PROGRAM BasketMemoryCtrl
VAR

	NIL: BOOL;

END_VAR

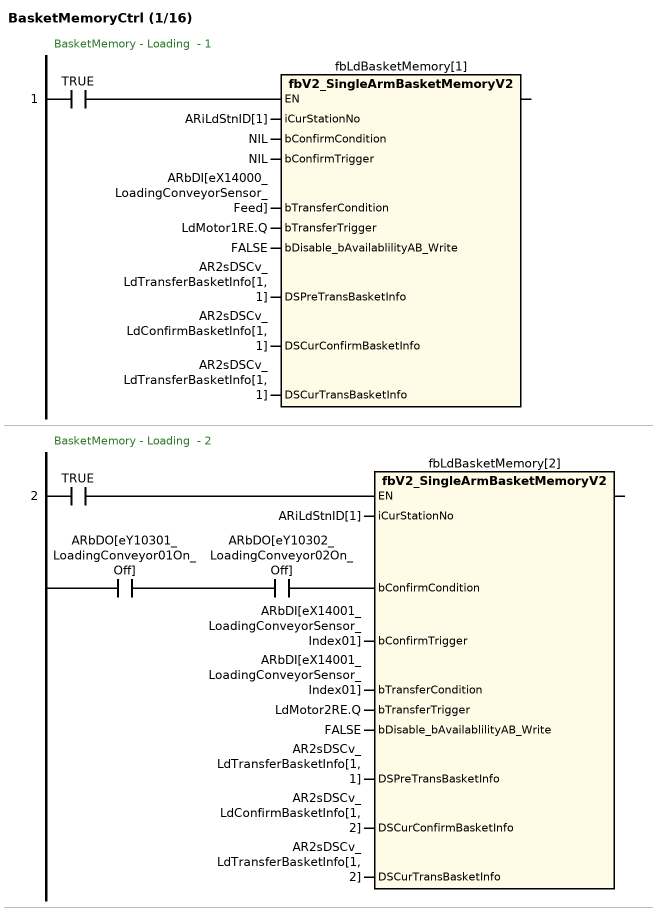
// NETWORK 1
// BasketMemory - Loading  - 1
fbLdBasketMemory[1](
    iCurStationNo := ARiLdStnID[1],
    bConfirmCondition := NIL,
    bConfirmTrigger := NIL,
    bTransferCondition := ARbDI[eX14000_LoadingConveyorSensor_Feed],
    bTransferTrigger := LdMotor1RE.Q,
    bDisable_bAvailablilityAB_Write := FALSE,
    DSPreTransBasketInfo := AR2sDSCv_LdTransferBasketInfo[1,1],
    DSCurConfirmBasketInfo := AR2sDSCv_LdConfirmBasketInfo[1,1],
    DSCurTransBasketInfo := AR2sDSCv_LdTransferBasketInfo[1,1]); // fbV2_SingleArmBasketMemoryV2

// NETWORK 2
// BasketMemory - Loading  - 2
fbLdBasketMemory[2](
    iCurStationNo := ARiLdStnID[1],
    bConfirmCondition := ARbDO[eY10301_LoadingConveyor01On_Off] AND ARbDO[eY10302_LoadingConveyor02On_Off],
    bConfirmTrigger := ARbDI[eX14001_LoadingConveyorSensor_Index01],
    bTransferCondition := ARbDI[eX14001_LoadingConveyorSensor_Index01],
    bTransferTrigger := LdMotor2RE.Q,
    bDisable_bAvailablilityAB_Write := FALSE,
    DSPreTransBasketInfo := AR2sDSCv_LdTransferBasketInfo[1,1],
    DSCurConfirmBasketInfo := AR2sDSCv_LdConfirmBasketInfo[1,2],
    DSCurTransBasketInfo := AR2sDSCv_LdTransferBasketInfo[1,2]); // fbV2_SingleArmBasketMemoryV2

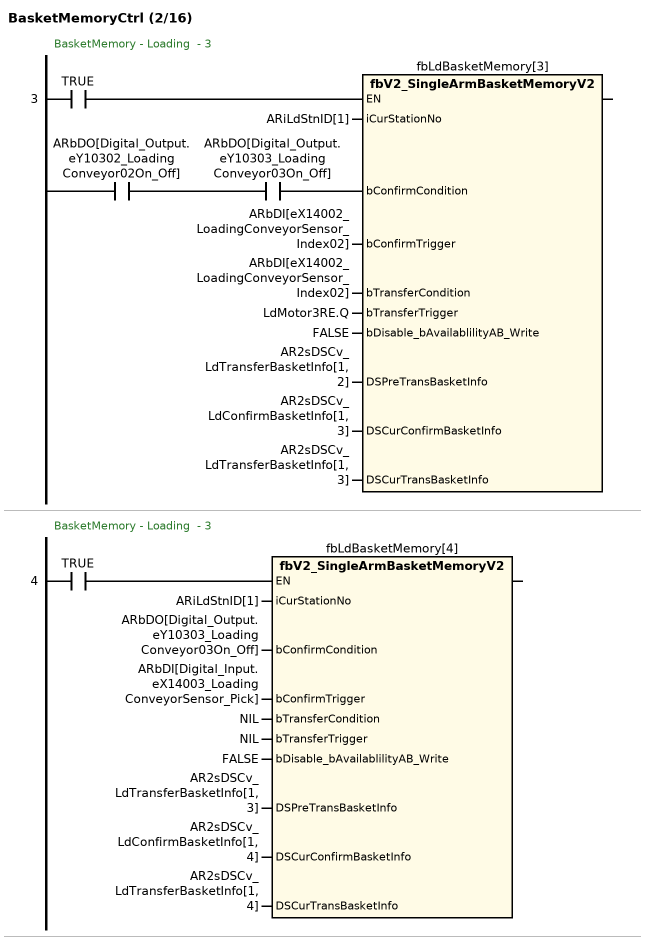
// NETWORK 3
// BasketMemory - Loading  - 3
fbLdBasketMemory[3](
    iCurStationNo := ARiLdStnID[1],
    bConfirmCondition := ARbDO[Digital_Output.eY10302_LoadingConveyor02On_Off] AND ARbDO[Digital_Output.eY10303_LoadingConveyor03On_Off],
    bConfirmTrigger := ARbDI[eX14002_LoadingConveyorSensor_Index02],
    bTransferCondition := ARbDI[eX14002_LoadingConveyorSensor_Index02],
    bTransferTrigger := LdMotor3RE.Q,
    bDisable_bAvailablilityAB_Write := FALSE,
    DSPreTransBasketInfo := AR2sDSCv_LdTransferBasketInfo[1,2],
    DSCurConfirmBasketInfo := AR2sDSCv_LdConfirmBasketInfo[1,3],
    DSCurTransBasketInfo := AR2sDSCv_LdTransferBasketInfo[1,3]); // fbV2_SingleArmBasketMemoryV2

// NETWORK 4
// BasketMemory - Loading  - 3
fbLdBasketMemory[4](
    iCurStationNo := ARiLdStnID[1],
    bConfirmCondition := ARbDO[Digital_Output.eY10303_LoadingConveyor03On_Off],
    bConfirmTrigger := ARbDI[Digital_Input.eX14003_LoadingConveyorSensor_Pick],
    bTransferCondition := NIL,
    bTransferTrigger := NIL,
    bDisable_bAvailablilityAB_Write := FALSE,
    DSPreTransBasketInfo := AR2sDSCv_LdTransferBasketInfo[1,3],
    DSCurConfirmBasketInfo := AR2sDSCv_LdConfirmBasketInfo[1,4],
    DSCurTransBasketInfo := AR2sDSCv_LdTransferBasketInfo[1,4]); // fbV2_SingleArmBasketMemoryV2

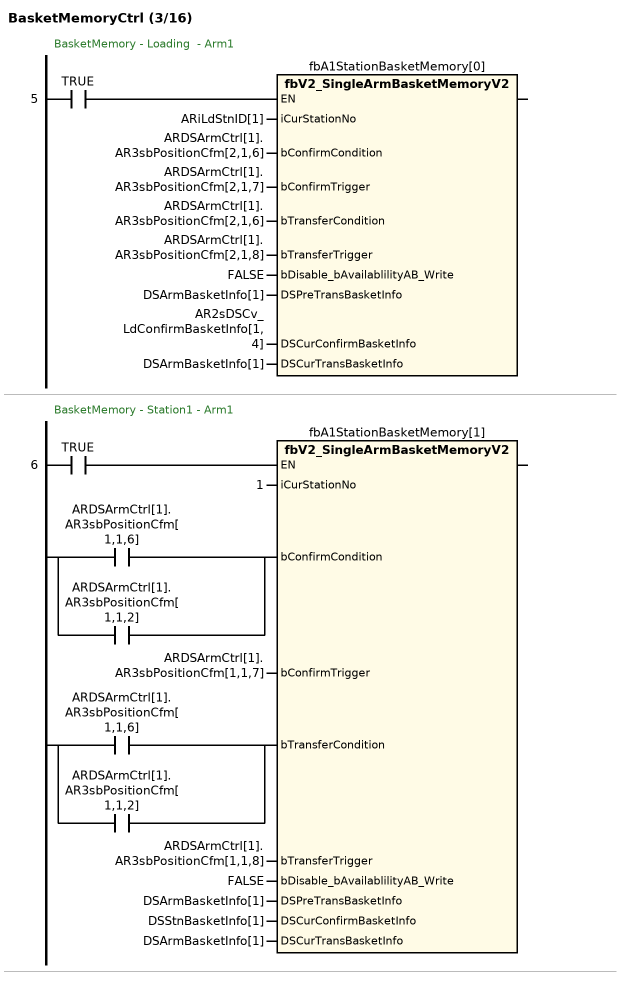
// NETWORK 5
// BasketMemory - Loading  - Arm1
fbA1StationBasketMemory[0](
    iCurStationNo := ARiLdStnID[1],
    bConfirmCondition := ARDSArmCtrl[1].AR3sbPositionCfm[2,1,6],
    bConfirmTrigger := ARDSArmCtrl[1].AR3sbPositionCfm[2,1,7],
    bTransferCondition := ARDSArmCtrl[1].AR3sbPositionCfm[2,1,6],
    bTransferTrigger := ARDSArmCtrl[1].AR3sbPositionCfm[2,1,8],
    bDisable_bAvailablilityAB_Write := FALSE,
    DSPreTransBasketInfo := DSArmBasketInfo[1],
    DSCurConfirmBasketInfo := AR2sDSCv_LdConfirmBasketInfo[1,4],
    DSCurTransBasketInfo := DSArmBasketInfo[1]); // fbV2_SingleArmBasketMemoryV2

// NETWORK 6
// BasketMemory - Station1 - Arm1
fbA1StationBasketMemory[1](
    iCurStationNo := 1,
    bConfirmCondition := ARDSArmCtrl[1].AR3sbPositionCfm[1,1,6] OR ARDSArmCtrl[1].AR3sbPositionCfm[1,1,2],
    bConfirmTrigger := ARDSArmCtrl[1].AR3sbPositionCfm[1,1,7],
    bTransferCondition := ARDSArmCtrl[1].AR3sbPositionCfm[1,1,6] OR ARDSArmCtrl[1].AR3sbPositionCfm[1,1,2],
    bTransferTrigger := ARDSArmCtrl[1].AR3sbPositionCfm[1,1,8],
    bDisable_bAvailablilityAB_Write := FALSE,
    DSPreTransBasketInfo := DSArmBasketInfo[1],
    DSCurConfirmBasketInfo := DSStnBasketInfo[1],
    DSCurTransBasketInfo := DSArmBasketInfo[1]); // fbV2_SingleArmBasketMemoryV2

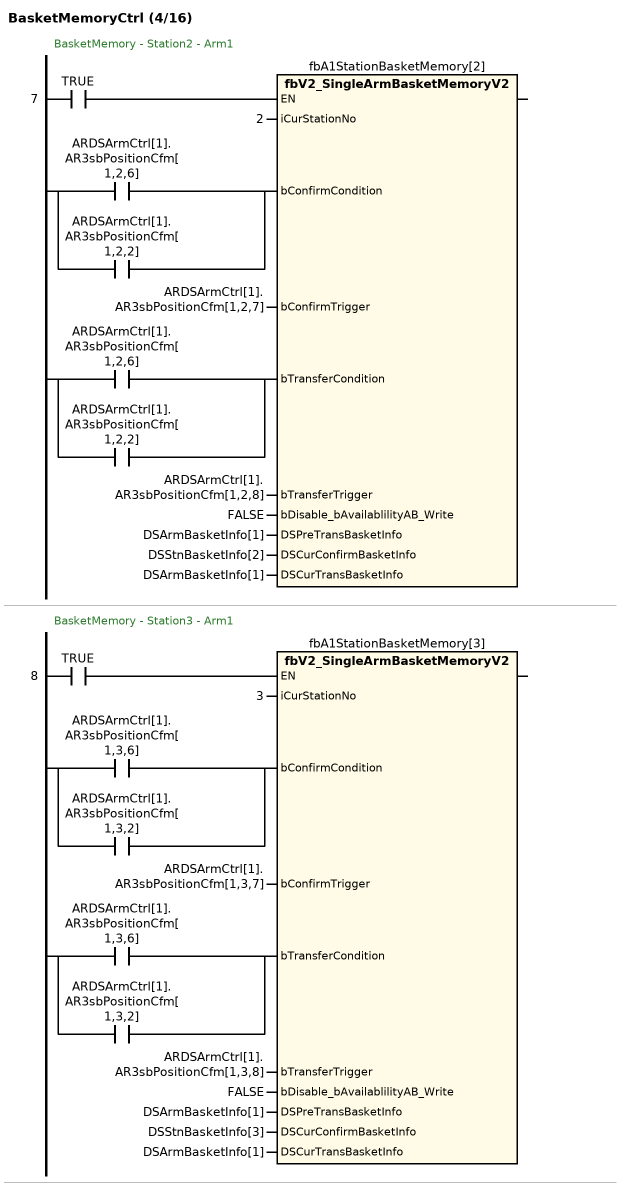
// NETWORK 7
// BasketMemory - Station2 - Arm1
fbA1StationBasketMemory[2](
    iCurStationNo := 2,
    bConfirmCondition := ARDSArmCtrl[1].AR3sbPositionCfm[1,2,6] OR ARDSArmCtrl[1].AR3sbPositionCfm[1,2,2],
    bConfirmTrigger := ARDSArmCtrl[1].AR3sbPositionCfm[1,2,7],
    bTransferCondition := ARDSArmCtrl[1].AR3sbPositionCfm[1,2,6] OR ARDSArmCtrl[1].AR3sbPositionCfm[1,2,2],
    bTransferTrigger := ARDSArmCtrl[1].AR3sbPositionCfm[1,2,8],
    bDisable_bAvailablilityAB_Write := FALSE,
    DSPreTransBasketInfo := DSArmBasketInfo[1],
    DSCurConfirmBasketInfo := DSStnBasketInfo[2],
    DSCurTransBasketInfo := DSArmBasketInfo[1]); // fbV2_SingleArmBasketMemoryV2

// NETWORK 8
// BasketMemory - Station3 - Arm1
fbA1StationBasketMemory[3](
    iCurStationNo := 3,
    bConfirmCondition := ARDSArmCtrl[1].AR3sbPositionCfm[1,3,6] OR ARDSArmCtrl[1].AR3sbPositionCfm[1,3,2],
    bConfirmTrigger := ARDSArmCtrl[1].AR3sbPositionCfm[1,3,7],
    bTransferCondition := ARDSArmCtrl[1].AR3sbPositionCfm[1,3,6] OR ARDSArmCtrl[1].AR3sbPositionCfm[1,3,2],
    bTransferTrigger := ARDSArmCtrl[1].AR3sbPositionCfm[1,3,8],
    bDisable_bAvailablilityAB_Write := FALSE,
    DSPreTransBasketInfo := DSArmBasketInfo[1],
    DSCurConfirmBasketInfo := DSStnBasketInfo[3],
    DSCurTransBasketInfo := DSArmBasketInfo[1]); // fbV2_SingleArmBasketMemoryV2

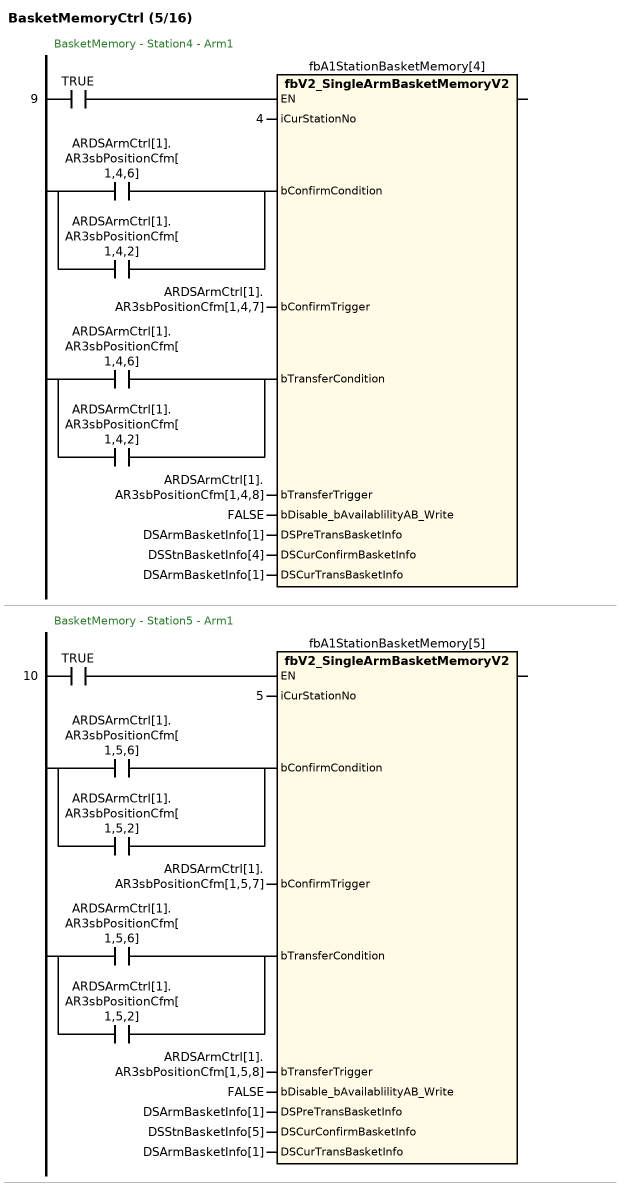
// NETWORK 9
// BasketMemory - Station4 - Arm1
fbA1StationBasketMemory[4](
    iCurStationNo := 4,
    bConfirmCondition := ARDSArmCtrl[1].AR3sbPositionCfm[1,4,6] OR ARDSArmCtrl[1].AR3sbPositionCfm[1,4,2],
    bConfirmTrigger := ARDSArmCtrl[1].AR3sbPositionCfm[1,4,7],
    bTransferCondition := ARDSArmCtrl[1].AR3sbPositionCfm[1,4,6] OR ARDSArmCtrl[1].AR3sbPositionCfm[1,4,2],
    bTransferTrigger := ARDSArmCtrl[1].AR3sbPositionCfm[1,4,8],
    bDisable_bAvailablilityAB_Write := FALSE,
    DSPreTransBasketInfo := DSArmBasketInfo[1],
    DSCurConfirmBasketInfo := DSStnBasketInfo[4],
    DSCurTransBasketInfo := DSArmBasketInfo[1]); // fbV2_SingleArmBasketMemoryV2

// NETWORK 10
// BasketMemory - Station5 - Arm1
fbA1StationBasketMemory[5](
    iCurStationNo := 5,
    bConfirmCondition := ARDSArmCtrl[1].AR3sbPositionCfm[1,5,6] OR ARDSArmCtrl[1].AR3sbPositionCfm[1,5,2],
    bConfirmTrigger := ARDSArmCtrl[1].AR3sbPositionCfm[1,5,7],
    bTransferCondition := ARDSArmCtrl[1].AR3sbPositionCfm[1,5,6] OR ARDSArmCtrl[1].AR3sbPositionCfm[1,5,2],
    bTransferTrigger := ARDSArmCtrl[1].AR3sbPositionCfm[1,5,8],
    bDisable_bAvailablilityAB_Write := FALSE,
    DSPreTransBasketInfo := DSArmBasketInfo[1],
    DSCurConfirmBasketInfo := DSStnBasketInfo[5],
    DSCurTransBasketInfo := DSArmBasketInfo[1]); // fbV2_SingleArmBasketMemoryV2

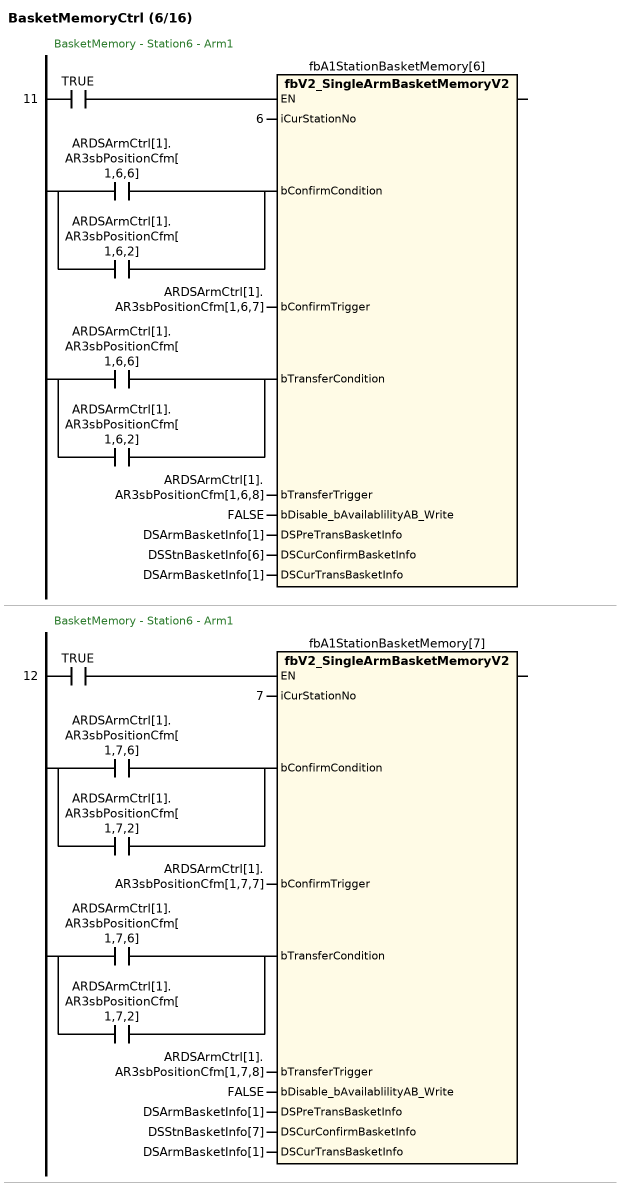
// NETWORK 11
// BasketMemory - Station6 - Arm1
fbA1StationBasketMemory[6](
    iCurStationNo := 6,
    bConfirmCondition := ARDSArmCtrl[1].AR3sbPositionCfm[1,6,6] OR ARDSArmCtrl[1].AR3sbPositionCfm[1,6,2],
    bConfirmTrigger := ARDSArmCtrl[1].AR3sbPositionCfm[1,6,7],
    bTransferCondition := ARDSArmCtrl[1].AR3sbPositionCfm[1,6,6] OR ARDSArmCtrl[1].AR3sbPositionCfm[1,6,2],
    bTransferTrigger := ARDSArmCtrl[1].AR3sbPositionCfm[1,6,8],
    bDisable_bAvailablilityAB_Write := FALSE,
    DSPreTransBasketInfo := DSArmBasketInfo[1],
    DSCurConfirmBasketInfo := DSStnBasketInfo[6],
    DSCurTransBasketInfo := DSArmBasketInfo[1]); // fbV2_SingleArmBasketMemoryV2

// NETWORK 12
// BasketMemory - Station6 - Arm1
fbA1StationBasketMemory[7](
    iCurStationNo := 7,
    bConfirmCondition := ARDSArmCtrl[1].AR3sbPositionCfm[1,7,6] OR ARDSArmCtrl[1].AR3sbPositionCfm[1,7,2],
    bConfirmTrigger := ARDSArmCtrl[1].AR3sbPositionCfm[1,7,7],
    bTransferCondition := ARDSArmCtrl[1].AR3sbPositionCfm[1,7,6] OR ARDSArmCtrl[1].AR3sbPositionCfm[1,7,2],
    bTransferTrigger := ARDSArmCtrl[1].AR3sbPositionCfm[1,7,8],
    bDisable_bAvailablilityAB_Write := FALSE,
    DSPreTransBasketInfo := DSArmBasketInfo[1],
    DSCurConfirmBasketInfo := DSStnBasketInfo[7],
    DSCurTransBasketInfo := DSArmBasketInfo[1]); // fbV2_SingleArmBasketMemoryV2

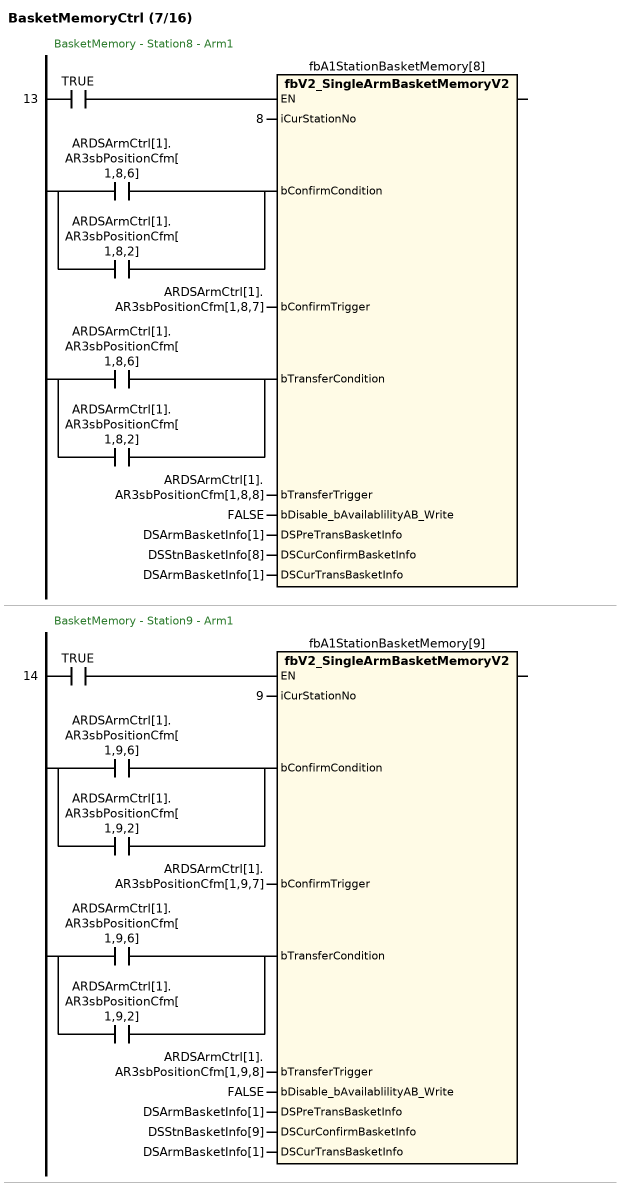
// NETWORK 13
// BasketMemory - Station8 - Arm1
fbA1StationBasketMemory[8](
    iCurStationNo := 8,
    bConfirmCondition := ARDSArmCtrl[1].AR3sbPositionCfm[1,8,6] OR ARDSArmCtrl[1].AR3sbPositionCfm[1,8,2],
    bConfirmTrigger := ARDSArmCtrl[1].AR3sbPositionCfm[1,8,7],
    bTransferCondition := ARDSArmCtrl[1].AR3sbPositionCfm[1,8,6] OR ARDSArmCtrl[1].AR3sbPositionCfm[1,8,2],
    bTransferTrigger := ARDSArmCtrl[1].AR3sbPositionCfm[1,8,8],
    bDisable_bAvailablilityAB_Write := FALSE,
    DSPreTransBasketInfo := DSArmBasketInfo[1],
    DSCurConfirmBasketInfo := DSStnBasketInfo[8],
    DSCurTransBasketInfo := DSArmBasketInfo[1]); // fbV2_SingleArmBasketMemoryV2

// NETWORK 14
// BasketMemory - Station9 - Arm1
fbA1StationBasketMemory[9](
    iCurStationNo := 9,
    bConfirmCondition := ARDSArmCtrl[1].AR3sbPositionCfm[1,9,6] OR ARDSArmCtrl[1].AR3sbPositionCfm[1,9,2],
    bConfirmTrigger := ARDSArmCtrl[1].AR3sbPositionCfm[1,9,7],
    bTransferCondition := ARDSArmCtrl[1].AR3sbPositionCfm[1,9,6] OR ARDSArmCtrl[1].AR3sbPositionCfm[1,9,2],
    bTransferTrigger := ARDSArmCtrl[1].AR3sbPositionCfm[1,9,8],
    bDisable_bAvailablilityAB_Write := FALSE,
    DSPreTransBasketInfo := DSArmBasketInfo[1],
    DSCurConfirmBasketInfo := DSStnBasketInfo[9],
    DSCurTransBasketInfo := DSArmBasketInfo[1]); // fbV2_SingleArmBasketMemoryV2

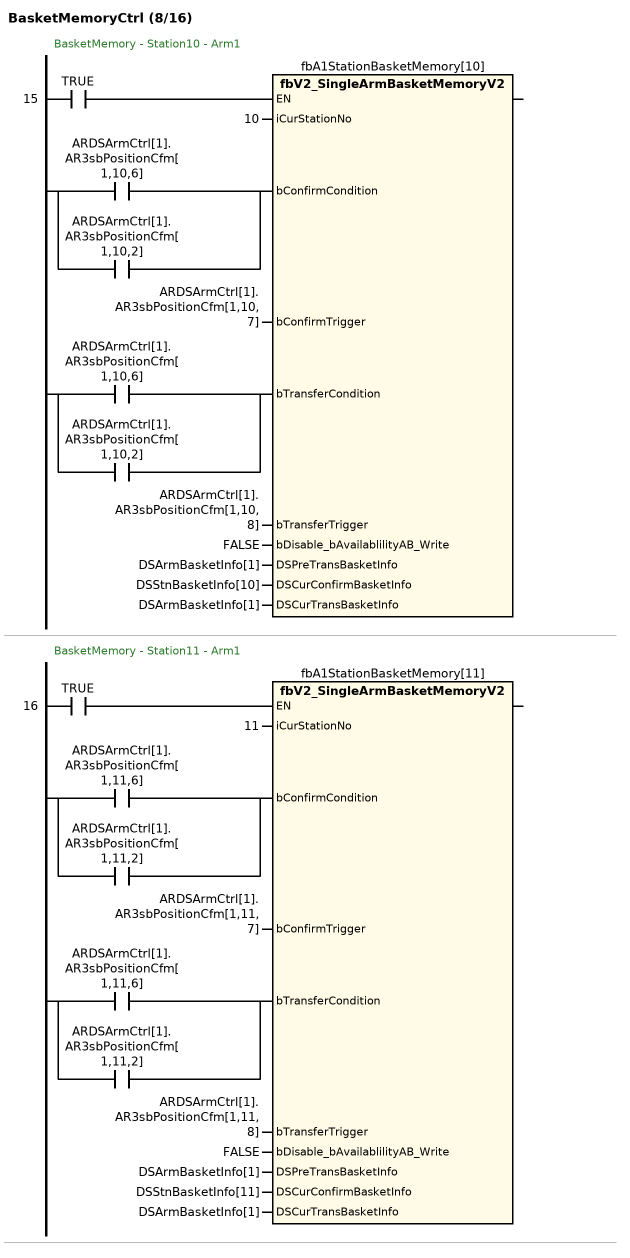
// NETWORK 15
// BasketMemory - Station10 - Arm1
fbA1StationBasketMemory[10](
    iCurStationNo := 10,
    bConfirmCondition := ARDSArmCtrl[1].AR3sbPositionCfm[1,10,6] OR ARDSArmCtrl[1].AR3sbPositionCfm[1,10,2],
    bConfirmTrigger := ARDSArmCtrl[1].AR3sbPositionCfm[1,10,7],
    bTransferCondition := ARDSArmCtrl[1].AR3sbPositionCfm[1,10,6] OR ARDSArmCtrl[1].AR3sbPositionCfm[1,10,2],
    bTransferTrigger := ARDSArmCtrl[1].AR3sbPositionCfm[1,10,8],
    bDisable_bAvailablilityAB_Write := FALSE,
    DSPreTransBasketInfo := DSArmBasketInfo[1],
    DSCurConfirmBasketInfo := DSStnBasketInfo[10],
    DSCurTransBasketInfo := DSArmBasketInfo[1]); // fbV2_SingleArmBasketMemoryV2

// NETWORK 16
// BasketMemory - Station11 - Arm1
fbA1StationBasketMemory[11](
    iCurStationNo := 11,
    bConfirmCondition := ARDSArmCtrl[1].AR3sbPositionCfm[1,11,6] OR ARDSArmCtrl[1].AR3sbPositionCfm[1,11,2],
    bConfirmTrigger := ARDSArmCtrl[1].AR3sbPositionCfm[1,11,7],
    bTransferCondition := ARDSArmCtrl[1].AR3sbPositionCfm[1,11,6] OR ARDSArmCtrl[1].AR3sbPositionCfm[1,11,2],
    bTransferTrigger := ARDSArmCtrl[1].AR3sbPositionCfm[1,11,8],
    bDisable_bAvailablilityAB_Write := FALSE,
    DSPreTransBasketInfo := DSArmBasketInfo[1],
    DSCurConfirmBasketInfo := DSStnBasketInfo[11],
    DSCurTransBasketInfo := DSArmBasketInfo[1]); // fbV2_SingleArmBasketMemoryV2

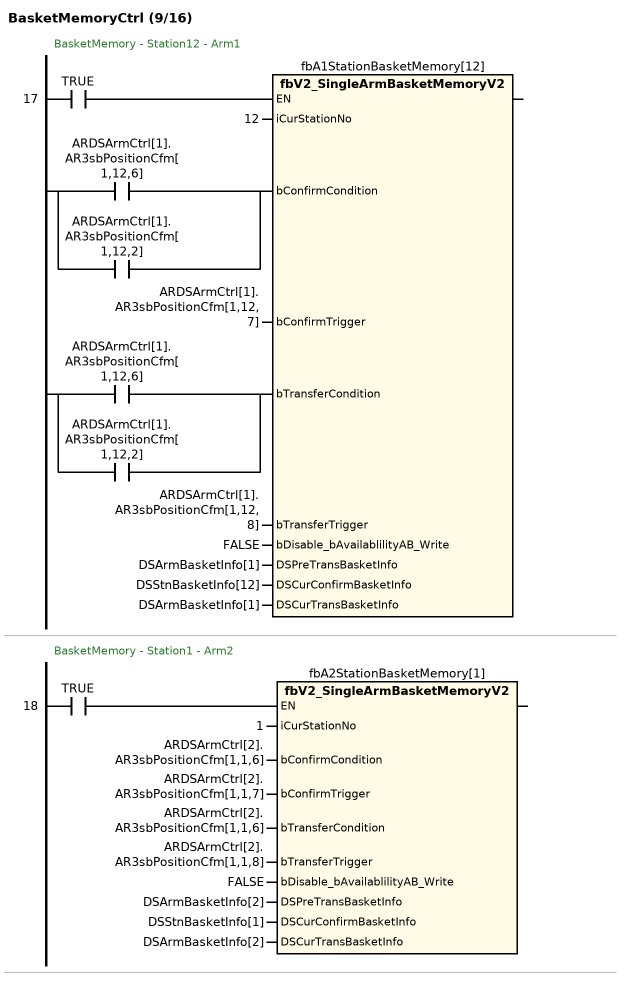
// NETWORK 17
// BasketMemory - Station12 - Arm1
fbA1StationBasketMemory[12](
    iCurStationNo := 12,
    bConfirmCondition := ARDSArmCtrl[1].AR3sbPositionCfm[1,12,6] OR ARDSArmCtrl[1].AR3sbPositionCfm[1,12,2],
    bConfirmTrigger := ARDSArmCtrl[1].AR3sbPositionCfm[1,12,7],
    bTransferCondition := ARDSArmCtrl[1].AR3sbPositionCfm[1,12,6] OR ARDSArmCtrl[1].AR3sbPositionCfm[1,12,2],
    bTransferTrigger := ARDSArmCtrl[1].AR3sbPositionCfm[1,12,8],
    bDisable_bAvailablilityAB_Write := FALSE,
    DSPreTransBasketInfo := DSArmBasketInfo[1],
    DSCurConfirmBasketInfo := DSStnBasketInfo[12],
    DSCurTransBasketInfo := DSArmBasketInfo[1]); // fbV2_SingleArmBasketMemoryV2

// NETWORK 18
// BasketMemory - Station1 - Arm2
fbA2StationBasketMemory[1](
    iCurStationNo := 1,
    bConfirmCondition := ARDSArmCtrl[2].AR3sbPositionCfm[1,1,6],
    bConfirmTrigger := ARDSArmCtrl[2].AR3sbPositionCfm[1,1,7],
    bTransferCondition := ARDSArmCtrl[2].AR3sbPositionCfm[1,1,6],
    bTransferTrigger := ARDSArmCtrl[2].AR3sbPositionCfm[1,1,8],
    bDisable_bAvailablilityAB_Write := FALSE,
    DSPreTransBasketInfo := DSArmBasketInfo[2],
    DSCurConfirmBasketInfo := DSStnBasketInfo[1],
    DSCurTransBasketInfo := DSArmBasketInfo[2]); // fbV2_SingleArmBasketMemoryV2

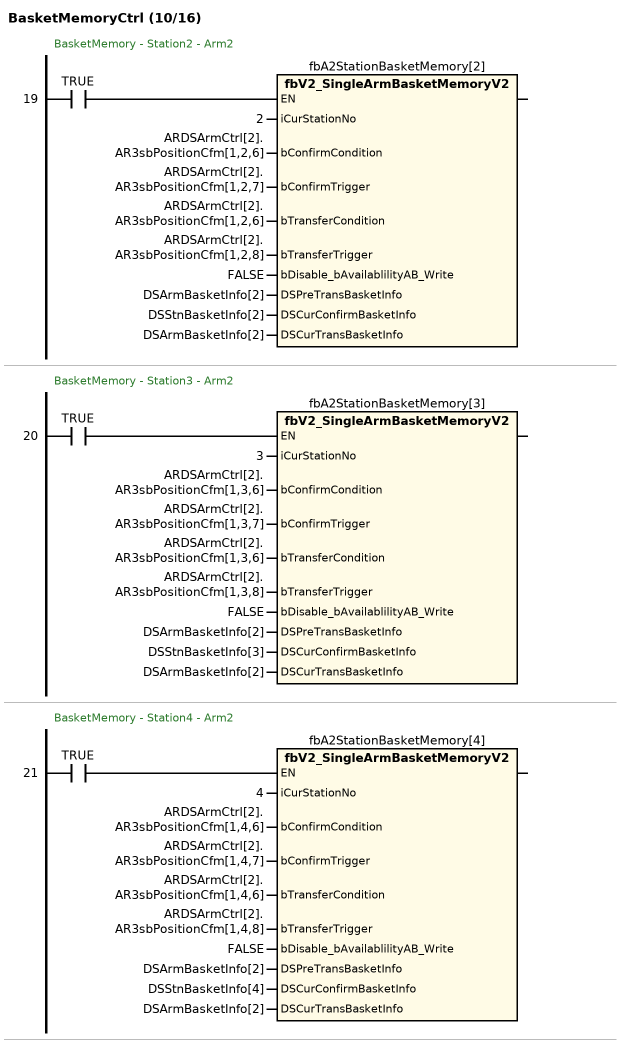
// NETWORK 19
// BasketMemory - Station2 - Arm2
fbA2StationBasketMemory[2](
    iCurStationNo := 2,
    bConfirmCondition := ARDSArmCtrl[2].AR3sbPositionCfm[1,2,6],
    bConfirmTrigger := ARDSArmCtrl[2].AR3sbPositionCfm[1,2,7],
    bTransferCondition := ARDSArmCtrl[2].AR3sbPositionCfm[1,2,6],
    bTransferTrigger := ARDSArmCtrl[2].AR3sbPositionCfm[1,2,8],
    bDisable_bAvailablilityAB_Write := FALSE,
    DSPreTransBasketInfo := DSArmBasketInfo[2],
    DSCurConfirmBasketInfo := DSStnBasketInfo[2],
    DSCurTransBasketInfo := DSArmBasketInfo[2]); // fbV2_SingleArmBasketMemoryV2

// NETWORK 20
// BasketMemory - Station3 - Arm2
fbA2StationBasketMemory[3](
    iCurStationNo := 3,
    bConfirmCondition := ARDSArmCtrl[2].AR3sbPositionCfm[1,3,6],
    bConfirmTrigger := ARDSArmCtrl[2].AR3sbPositionCfm[1,3,7],
    bTransferCondition := ARDSArmCtrl[2].AR3sbPositionCfm[1,3,6],
    bTransferTrigger := ARDSArmCtrl[2].AR3sbPositionCfm[1,3,8],
    bDisable_bAvailablilityAB_Write := FALSE,
    DSPreTransBasketInfo := DSArmBasketInfo[2],
    DSCurConfirmBasketInfo := DSStnBasketInfo[3],
    DSCurTransBasketInfo := DSArmBasketInfo[2]); // fbV2_SingleArmBasketMemoryV2

// NETWORK 21
// BasketMemory - Station4 - Arm2
fbA2StationBasketMemory[4](
    iCurStationNo := 4,
    bConfirmCondition := ARDSArmCtrl[2].AR3sbPositionCfm[1,4,6],
    bConfirmTrigger := ARDSArmCtrl[2].AR3sbPositionCfm[1,4,7],
    bTransferCondition := ARDSArmCtrl[2].AR3sbPositionCfm[1,4,6],
    bTransferTrigger := ARDSArmCtrl[2].AR3sbPositionCfm[1,4,8],
    bDisable_bAvailablilityAB_Write := FALSE,
    DSPreTransBasketInfo := DSArmBasketInfo[2],
    DSCurConfirmBasketInfo := DSStnBasketInfo[4],
    DSCurTransBasketInfo := DSArmBasketInfo[2]); // fbV2_SingleArmBasketMemoryV2

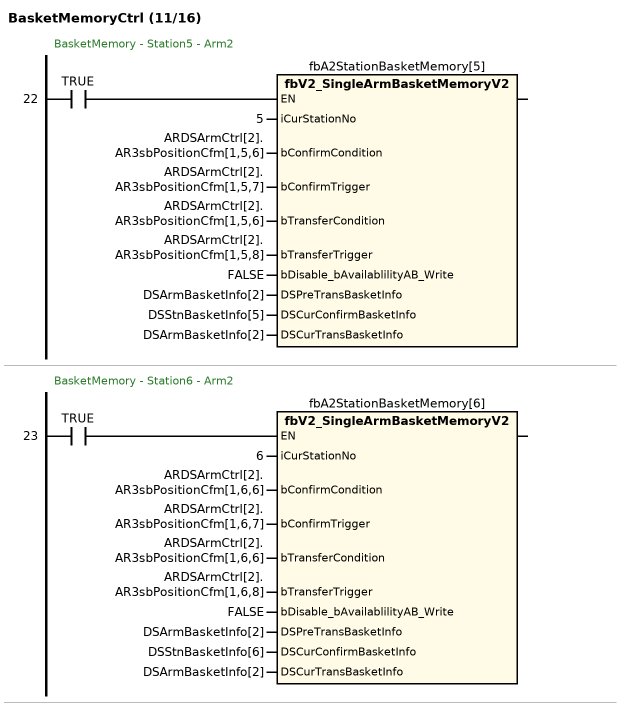
// NETWORK 22
// BasketMemory - Station5 - Arm2
fbA2StationBasketMemory[5](
    iCurStationNo := 5,
    bConfirmCondition := ARDSArmCtrl[2].AR3sbPositionCfm[1,5,6],
    bConfirmTrigger := ARDSArmCtrl[2].AR3sbPositionCfm[1,5,7],
    bTransferCondition := ARDSArmCtrl[2].AR3sbPositionCfm[1,5,6],
    bTransferTrigger := ARDSArmCtrl[2].AR3sbPositionCfm[1,5,8],
    bDisable_bAvailablilityAB_Write := FALSE,
    DSPreTransBasketInfo := DSArmBasketInfo[2],
    DSCurConfirmBasketInfo := DSStnBasketInfo[5],
    DSCurTransBasketInfo := DSArmBasketInfo[2]); // fbV2_SingleArmBasketMemoryV2

// NETWORK 23
// BasketMemory - Station6 - Arm2
fbA2StationBasketMemory[6](
    iCurStationNo := 6,
    bConfirmCondition := ARDSArmCtrl[2].AR3sbPositionCfm[1,6,6],
    bConfirmTrigger := ARDSArmCtrl[2].AR3sbPositionCfm[1,6,7],
    bTransferCondition := ARDSArmCtrl[2].AR3sbPositionCfm[1,6,6],
    bTransferTrigger := ARDSArmCtrl[2].AR3sbPositionCfm[1,6,8],
    bDisable_bAvailablilityAB_Write := FALSE,
    DSPreTransBasketInfo := DSArmBasketInfo[2],
    DSCurConfirmBasketInfo := DSStnBasketInfo[6],
    DSCurTransBasketInfo := DSArmBasketInfo[2]); // fbV2_SingleArmBasketMemoryV2

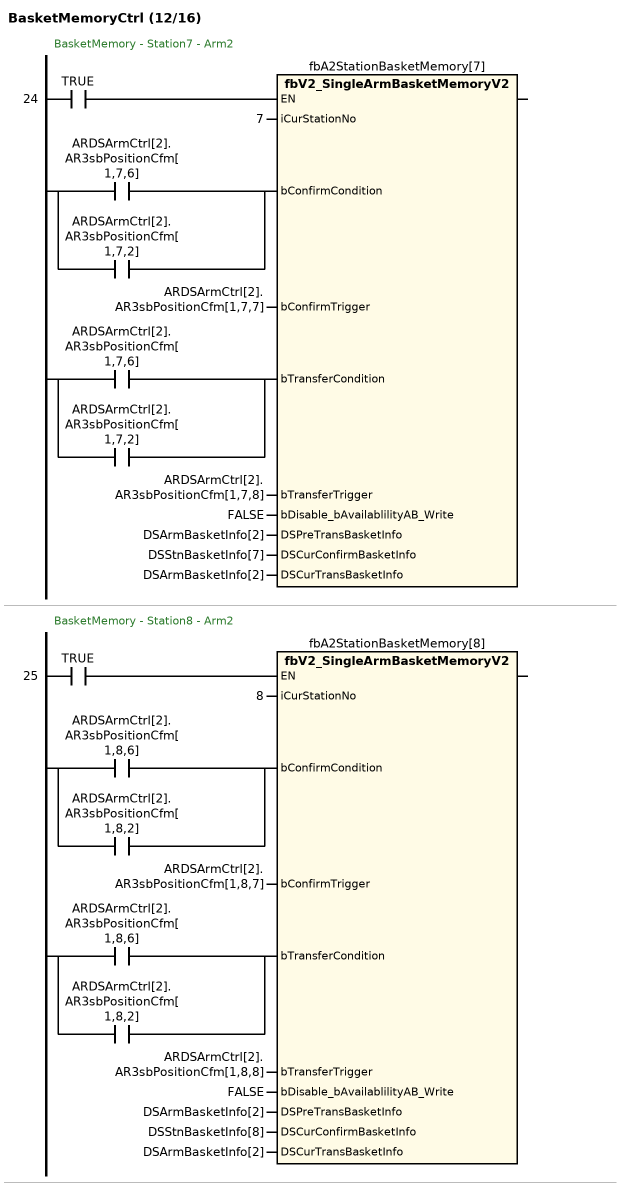
// NETWORK 24
// BasketMemory - Station7 - Arm2
fbA2StationBasketMemory[7](
    iCurStationNo := 7,
    bConfirmCondition := ARDSArmCtrl[2].AR3sbPositionCfm[1,7,6] OR ARDSArmCtrl[2].AR3sbPositionCfm[1,7,2],
    bConfirmTrigger := ARDSArmCtrl[2].AR3sbPositionCfm[1,7,7],
    bTransferCondition := ARDSArmCtrl[2].AR3sbPositionCfm[1,7,6] OR ARDSArmCtrl[2].AR3sbPositionCfm[1,7,2],
    bTransferTrigger := ARDSArmCtrl[2].AR3sbPositionCfm[1,7,8],
    bDisable_bAvailablilityAB_Write := FALSE,
    DSPreTransBasketInfo := DSArmBasketInfo[2],
    DSCurConfirmBasketInfo := DSStnBasketInfo[7],
    DSCurTransBasketInfo := DSArmBasketInfo[2]); // fbV2_SingleArmBasketMemoryV2

// NETWORK 25
// BasketMemory - Station8 - Arm2
fbA2StationBasketMemory[8](
    iCurStationNo := 8,
    bConfirmCondition := ARDSArmCtrl[2].AR3sbPositionCfm[1,8,6] OR ARDSArmCtrl[2].AR3sbPositionCfm[1,8,2],
    bConfirmTrigger := ARDSArmCtrl[2].AR3sbPositionCfm[1,8,7],
    bTransferCondition := ARDSArmCtrl[2].AR3sbPositionCfm[1,8,6] OR ARDSArmCtrl[2].AR3sbPositionCfm[1,8,2],
    bTransferTrigger := ARDSArmCtrl[2].AR3sbPositionCfm[1,8,8],
    bDisable_bAvailablilityAB_Write := FALSE,
    DSPreTransBasketInfo := DSArmBasketInfo[2],
    DSCurConfirmBasketInfo := DSStnBasketInfo[8],
    DSCurTransBasketInfo := DSArmBasketInfo[2]); // fbV2_SingleArmBasketMemoryV2

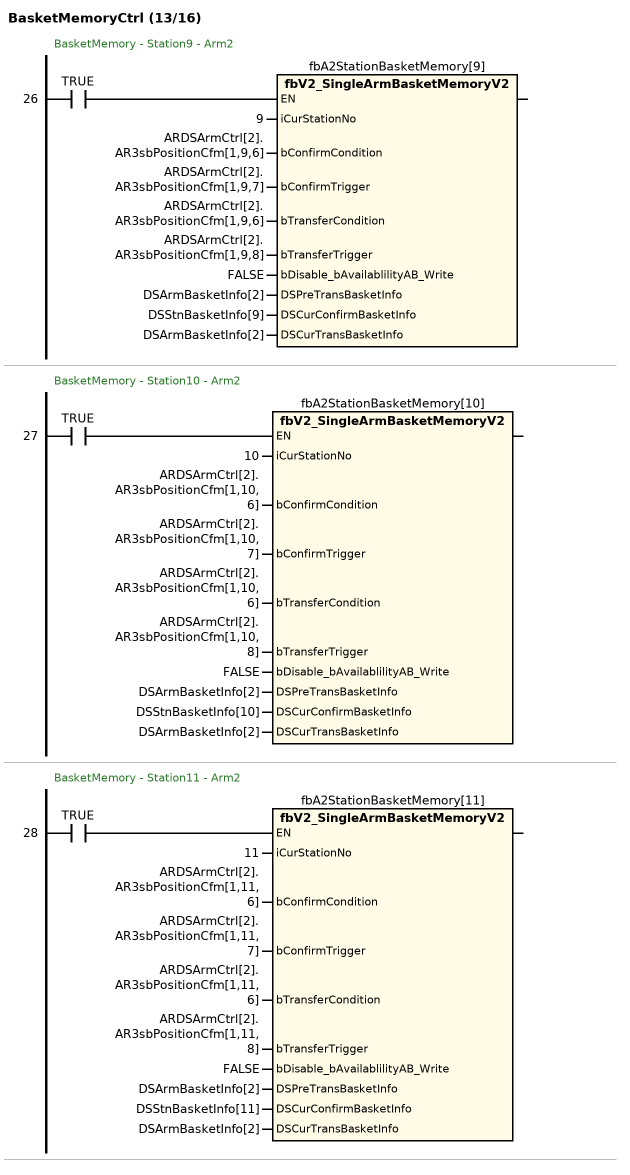
// NETWORK 26
// BasketMemory - Station9 - Arm2
fbA2StationBasketMemory[9](
    iCurStationNo := 9,
    bConfirmCondition := ARDSArmCtrl[2].AR3sbPositionCfm[1,9,6],
    bConfirmTrigger := ARDSArmCtrl[2].AR3sbPositionCfm[1,9,7],
    bTransferCondition := ARDSArmCtrl[2].AR3sbPositionCfm[1,9,6],
    bTransferTrigger := ARDSArmCtrl[2].AR3sbPositionCfm[1,9,8],
    bDisable_bAvailablilityAB_Write := FALSE,
    DSPreTransBasketInfo := DSArmBasketInfo[2],
    DSCurConfirmBasketInfo := DSStnBasketInfo[9],
    DSCurTransBasketInfo := DSArmBasketInfo[2]); // fbV2_SingleArmBasketMemoryV2

// NETWORK 27
// BasketMemory - Station10 - Arm2
fbA2StationBasketMemory[10](
    iCurStationNo := 10,
    bConfirmCondition := ARDSArmCtrl[2].AR3sbPositionCfm[1,10,6],
    bConfirmTrigger := ARDSArmCtrl[2].AR3sbPositionCfm[1,10,7],
    bTransferCondition := ARDSArmCtrl[2].AR3sbPositionCfm[1,10,6],
    bTransferTrigger := ARDSArmCtrl[2].AR3sbPositionCfm[1,10,8],
    bDisable_bAvailablilityAB_Write := FALSE,
    DSPreTransBasketInfo := DSArmBasketInfo[2],
    DSCurConfirmBasketInfo := DSStnBasketInfo[10],
    DSCurTransBasketInfo := DSArmBasketInfo[2]); // fbV2_SingleArmBasketMemoryV2

// NETWORK 28
// BasketMemory - Station11 - Arm2
fbA2StationBasketMemory[11](
    iCurStationNo := 11,
    bConfirmCondition := ARDSArmCtrl[2].AR3sbPositionCfm[1,11,6],
    bConfirmTrigger := ARDSArmCtrl[2].AR3sbPositionCfm[1,11,7],
    bTransferCondition := ARDSArmCtrl[2].AR3sbPositionCfm[1,11,6],
    bTransferTrigger := ARDSArmCtrl[2].AR3sbPositionCfm[1,11,8],
    bDisable_bAvailablilityAB_Write := FALSE,
    DSPreTransBasketInfo := DSArmBasketInfo[2],
    DSCurConfirmBasketInfo := DSStnBasketInfo[11],
    DSCurTransBasketInfo := DSArmBasketInfo[2]); // fbV2_SingleArmBasketMemoryV2

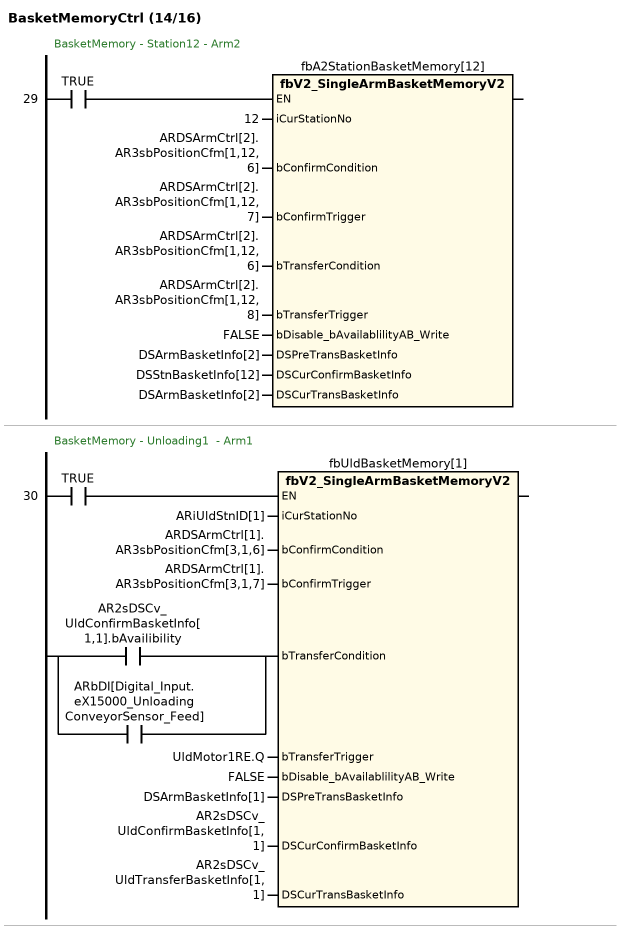
// NETWORK 29
// BasketMemory - Station12 - Arm2
fbA2StationBasketMemory[12](
    iCurStationNo := 12,
    bConfirmCondition := ARDSArmCtrl[2].AR3sbPositionCfm[1,12,6],
    bConfirmTrigger := ARDSArmCtrl[2].AR3sbPositionCfm[1,12,7],
    bTransferCondition := ARDSArmCtrl[2].AR3sbPositionCfm[1,12,6],
    bTransferTrigger := ARDSArmCtrl[2].AR3sbPositionCfm[1,12,8],
    bDisable_bAvailablilityAB_Write := FALSE,
    DSPreTransBasketInfo := DSArmBasketInfo[2],
    DSCurConfirmBasketInfo := DSStnBasketInfo[12],
    DSCurTransBasketInfo := DSArmBasketInfo[2]); // fbV2_SingleArmBasketMemoryV2

// NETWORK 30
// BasketMemory - Unloading1  - Arm1
fbUldBasketMemory[1](
    iCurStationNo := ARiUldStnID[1],
    bConfirmCondition := ARDSArmCtrl[1].AR3sbPositionCfm[3,1,6],
    bConfirmTrigger := ARDSArmCtrl[1].AR3sbPositionCfm[3,1,7],
    bTransferCondition := AR2sDSCv_UldConfirmBasketInfo[1,1].bAvailibility OR ARbDI[Digital_Input.eX15000_UnloadingConveyorSensor_Feed],
    bTransferTrigger := UldMotor1RE.Q,
    bDisable_bAvailablilityAB_Write := FALSE,
    DSPreTransBasketInfo := DSArmBasketInfo[1],
    DSCurConfirmBasketInfo := AR2sDSCv_UldConfirmBasketInfo[1,1],
    DSCurTransBasketInfo := AR2sDSCv_UldTransferBasketInfo[1,1]); // fbV2_SingleArmBasketMemoryV2

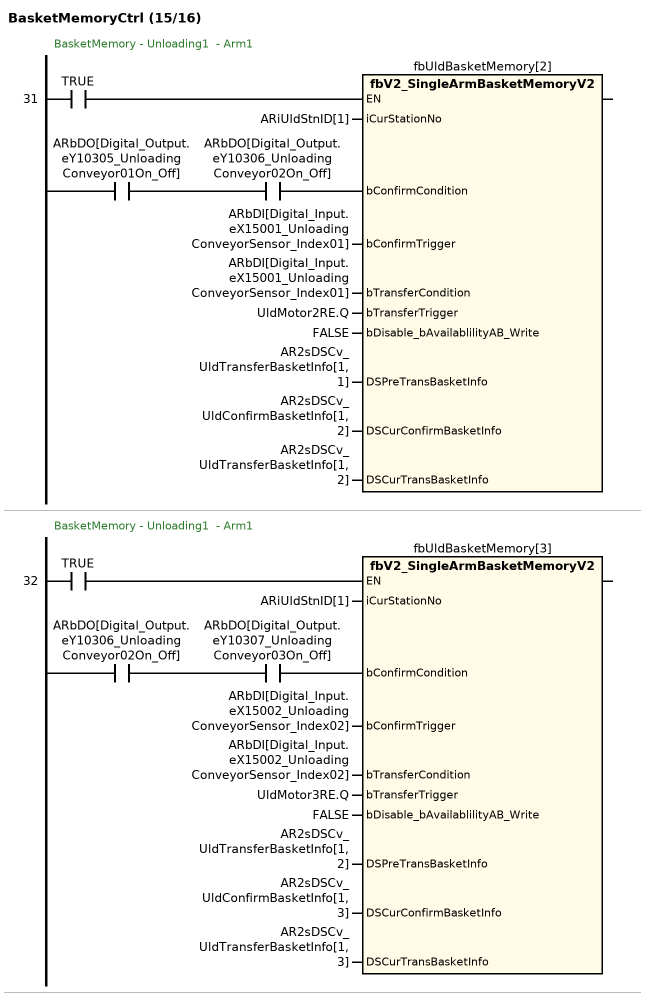
// NETWORK 31
// BasketMemory - Unloading1  - Arm1
fbUldBasketMemory[2](
    iCurStationNo := ARiUldStnID[1],
    bConfirmCondition := ARbDO[Digital_Output.eY10305_UnloadingConveyor01On_Off] AND ARbDO[Digital_Output.eY10306_UnloadingConveyor02On_Off],
    bConfirmTrigger := ARbDI[Digital_Input.eX15001_UnloadingConveyorSensor_Index01],
    bTransferCondition := ARbDI[Digital_Input.eX15001_UnloadingConveyorSensor_Index01],
    bTransferTrigger := UldMotor2RE.Q,
    bDisable_bAvailablilityAB_Write := FALSE,
    DSPreTransBasketInfo := AR2sDSCv_UldTransferBasketInfo[1,1],
    DSCurConfirmBasketInfo := AR2sDSCv_UldConfirmBasketInfo[1,2],
    DSCurTransBasketInfo := AR2sDSCv_UldTransferBasketInfo[1,2]); // fbV2_SingleArmBasketMemoryV2

// NETWORK 32
// BasketMemory - Unloading1  - Arm1
fbUldBasketMemory[3](
    iCurStationNo := ARiUldStnID[1],
    bConfirmCondition := ARbDO[Digital_Output.eY10306_UnloadingConveyor02On_Off] AND ARbDO[Digital_Output.eY10307_UnloadingConveyor03On_Off],
    bConfirmTrigger := ARbDI[Digital_Input.eX15002_UnloadingConveyorSensor_Index02],
    bTransferCondition := ARbDI[Digital_Input.eX15002_UnloadingConveyorSensor_Index02],
    bTransferTrigger := UldMotor3RE.Q,
    bDisable_bAvailablilityAB_Write := FALSE,
    DSPreTransBasketInfo := AR2sDSCv_UldTransferBasketInfo[1,2],
    DSCurConfirmBasketInfo := AR2sDSCv_UldConfirmBasketInfo[1,3],
    DSCurTransBasketInfo := AR2sDSCv_UldTransferBasketInfo[1,3]); // fbV2_SingleArmBasketMemoryV2

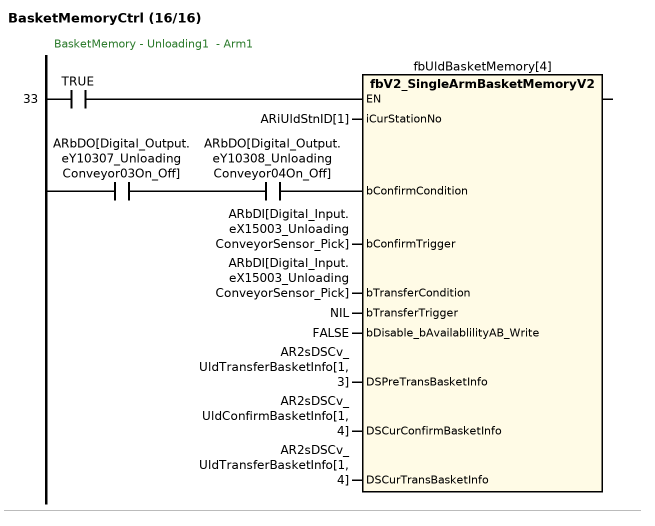
// NETWORK 33
// BasketMemory - Unloading1  - Arm1
fbUldBasketMemory[4](
    iCurStationNo := ARiUldStnID[1],
    bConfirmCondition := ARbDO[Digital_Output.eY10307_UnloadingConveyor03On_Off] AND ARbDO[Digital_Output.eY10308_UnloadingConveyor04On_Off],
    bConfirmTrigger := ARbDI[Digital_Input.eX15003_UnloadingConveyorSensor_Pick],
    bTransferCondition := ARbDI[Digital_Input.eX15003_UnloadingConveyorSensor_Pick],
    bTransferTrigger := NIL,
    bDisable_bAvailablilityAB_Write := FALSE,
    DSPreTransBasketInfo := AR2sDSCv_UldTransferBasketInfo[1,3],
    DSCurConfirmBasketInfo := AR2sDSCv_UldConfirmBasketInfo[1,4],
    DSCurTransBasketInfo := AR2sDSCv_UldTransferBasketInfo[1,4]); // fbV2_SingleArmBasketMemoryV2

END_PROGRAM

(* stored: Version 1.1.0.1, ProductVersion 3.1.4024.12
   POU BasketMemoryCtrl: Id {b6dff639-4b7a-4171-86e1-8c0ee3f1044c}, SpecialFunc None *)
